Fanuc KAREL source: KT00238.KL

PROGRAM KT00238
%NOLOCKGROUP
VAR
  I1: INTEGER
  Y2: ARRAY[2] OF BYTE
  OUT: INTEGER
BEGIN
  I1 = 2
    Y2[1] = 3
  OUT = I1 OR Y2[1]
END KT00238
